TYPE DUT_HMI EXTENDS DUT_Control_Base :
STRUCT
	AutoOn :BOOL;
	AutoOff :BOOL;
	ManualOn :BOOL;
	ManualOff :BOOL;
	ModeValue : INT:= 1; // 0: Manual; 1: Auto; 2: Interlock
END_STRUCT
END_TYPE

(* stored: Version 1.1.0.1, ProductVersion 3.1.4024.12
   DUT DUT_HMI: Id {7e2b4294-76ca-47d6-8c7b-fda0034aae6c} *)
